Omron CX-Programmer project NewProject (CX-Programmer 9.73)

# PLC NewPLC1: CP1E N20

## Global symbols (name address type ; comment)
0.00 BOOL  ; SUIS
100.00 BOOL  ; LAMP1
100.01 BOOL  ; LAMP 1
100.02 BOOL  ; LAMP2
T001 BOOL  ; TIMER 1
T002 BOOL  ; TIMER 2

## Program NewProgram1 (cyclic task 0)

### Section Section1

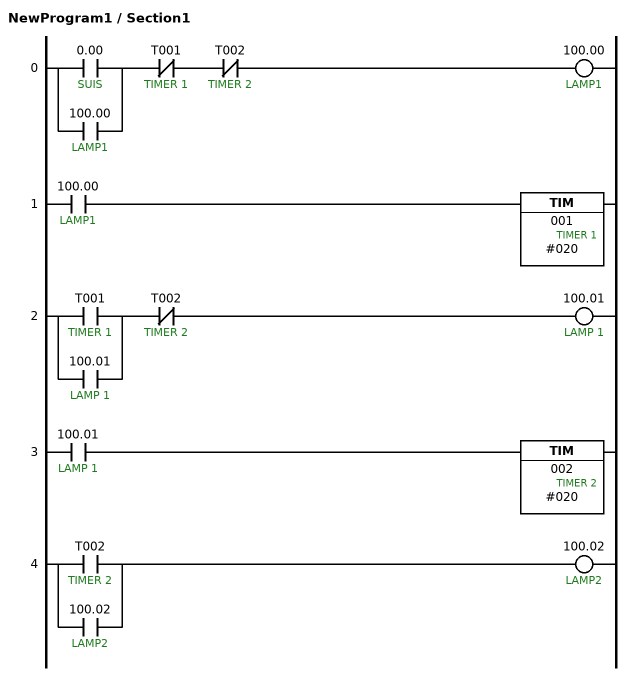
; rung 0
LD 0.00  ; SUIS
OR 100.00  ; LAMP1
ANDNOT T001  ; TIMER 1
ANDNOT T002  ; TIMER 2
OUT 100.00  ; LAMP1
; rung 1
LD 100.00  ; LAMP1
TIM 001 #020  ; TIMER 1
; rung 2
LD T001  ; TIMER 1
OR 100.01  ; LAMP 1
ANDNOT T002  ; TIMER 2
OUT 100.01  ; LAMP 1
; rung 3
LD 100.01  ; LAMP 1
TIM 002 #020  ; TIMER 2
; rung 4
LD T002  ; TIMER 2
OR 100.02  ; LAMP2
OUT 100.02  ; LAMP2

### Section END
; rung 0
END(001)